//{attribute 'qualified_only'}
VAR_GLOBAL
	b1stShot			: BOOL := TRUE;
	bPlcInitDone,
	bSettingsSaved		: BOOL;
	
	ILog				: I_Logger;
	fbEventHandler		: FB_EventHandler;
	
	fbRecipeManager		: FB_RecipeManager;
	fbVar2File			: FB_Var2File;
	stGlobalModuleInfo	: ST_MODULES_INFO; // global module/staion info
END_VAR
VAR_GLOBAL PERSISTENT
	// current system/machine configuration
	stConfig 			: ST_Configuration;
	
	// settings/recipe            
	stSettings			: ST_Settings;
	
	// PLC app system info
	stPlcAppSystemInfo	: PlcAppSystemInfo;
END_VAR

(* stored: Version 1.1.0.1
   GVL Services: Id {b0be6550-2810-4ccc-9dc7-dd711b7b0fac} *)
